FUNCTION F_Any_To_Generic : T_Generic
VAR_INPUT
	Value : ANY;
END_VAR

F_Any_To_Generic := Value;

END_FUNCTION

(* stored: Version 1.1.0.1
   POU F_Any_To_Generic: Id {70886885-63aa-0fec-045b-eb312a165e94}, SpecialFunc None *)
